// Mitsubishi GX Works2 project: 241010_비금석통과금석배출   PLC: Q03UDV

PROGRAM MAIN
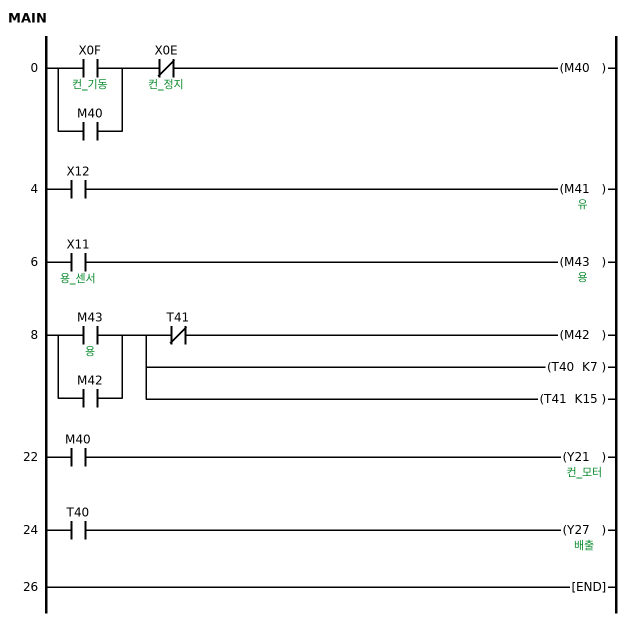
0     LD      X0F  ; 컨_기동
      OR      M40
      ANI     X0E  ; 컨_정지
      OUT     M40
4     LD      X12
      OUT     M41  ; 유
6     LD      X11  ; 용_센서
      OUT     M43  ; 용
8     LD      M43  ; 용
      OR      M42
      MPS
      ANI     T41
      OUT     M42
      MPP
      OUT     T40 K7
      OUT     T41 K15
22    LD      M40
      OUT     Y21  ; 컨_모터
24    LD      T40
      OUT     Y27  ; 배출
26    END
END_PROGRAM
